{attribute addProperty BoxType "EPP1258-0001-0016"}
{attribute addProperty Id "ChannelAT %I*ARRAY[0..7] OF Channel_E4AEF59E6480LatchAT %I*Latch_54D9ECC2272340WcStateAT %I*WcState_DC9C971540.50InfoDataAT %I*InfoData_7231B2DD80100"}
{attribute addProperty CRC "3998753854"}
{attribute addProperty SizeInBites "420"}
{attribute addProperty SizeInBytes "52.5"}
TYPE EPP1258_BB8E9A10 :
STRUCT
	{attribute addProperty Name "Channel"}
	Channel : ARRAY[0..7] OF Channel_E4AEF59E;
	{attribute addProperty Name "Latch"}
	Latch : Latch_54D9ECC2;
	{attribute addProperty Name "WcState"}
	WcState : WcState_DC9C9715;
	{attribute addProperty Name "InfoData"}
	InfoData : InfoData_7231B2DD;
END_STRUCT
END_TYPE

(* stored: Version 1.2.0.0, ProductVersion 3.1.4024.9
   DUT EPP1258_BB8E9A10: Id {dc9bc8de-e287-4e17-8f5f-8c25e6578899} *)
